{attribute addProperty BoxType "EL3356-0000-0017"}
{attribute addProperty Id "StatusAT %I*Status_42ED8037162"}
{attribute addProperty CRC "634153654"}
{attribute addProperty SizeInBites "16"}
{attribute addProperty SizeInBytes "2"}
TYPE RMB_Status_25CC6AB6 :
STRUCT
	{attribute addProperty Name "Status"}
	Status AT %I* : Status_42ED8037;
END_STRUCT
END_TYPE

(* stored: Version 1.2.0.0, ProductVersion 3.1.4024.9
   DUT RMB_Status_25CC6AB6: Id {17943a8a-7441-423b-b306-59d9ecd4d7b2} *)
